{attribute 'linkalways'} 
{attribute 'no_explicit_call' := 'This FB is a CLASS and must be accessed using methods or properties'}
{attribute 'enable_dynamic_creation'}
FUNCTION_BLOCK ABSTRACT NumericDatatypeBase EXTENDS DatatypeBase IMPLEMENTS I_NumericDatatype
VAR
END_VAR

PROPERTY PUBLIC ABSTRACT IsEven : BOOL
GET
END_GET
END_PROPERTY

PROPERTY PUBLIC ABSTRACT IsFloat : BOOL
GET
END_GET
END_PROPERTY

PROPERTY PUBLIC IsOdd : BOOL
GET
IsOdd := not IsEven;
END_GET
END_PROPERTY

PROPERTY PUBLIC ABSTRACT IsSigned : BOOL
GET
END_GET
END_PROPERTY

METHOD PROTECTED OnSerializeTypeWith
VAR_INPUT
	Serializer : I_Serializer;
END_VAR
SUPER^.OnSerializeTypeWith(Serializer);
Serializer.AddKey('minValue');
SerializeMinValue(Serializer);
Serializer.AddKey('maxValue');
SerializeMaxValue(Serializer);
Serializer.AddKeyBool('isSigned', IsSigned);
Serializer.AddKeyBool('isFloat', IsFloat);
END_METHOD

METHOD PROTECTED ABSTRACT SerializeMaxValue
VAR_INPUT
	Serializer : I_Serializer;
END_VAR
END_METHOD

METHOD PROTECTED ABSTRACT SerializeMinValue
VAR_INPUT
	Serializer : I_Serializer;
END_VAR
END_METHOD

END_FUNCTION_BLOCK

(* stored: Version 1.1.0.1, ProductVersion 3.1.4024.13
   POU NumericDatatypeBase: Id {96cfe585-e451-066a-0b8c-26079dae1329}, SpecialFunc None
   Folder Protected: Id {39e73c2d-fc59-01cc-09ba-b5d6d4e55439}
   Property IsEven: Id {f8cc3dde-0e09-0921-2005-35a3a6549198}
   Get Get: Id {ea3f34a8-8bb3-0245-0192-066a15b142d3}
   Property IsFloat: Id {db9b3e2c-dfd9-0457-2028-dc261a7bc18d}
   Get Get: Id {b25b2249-b422-0a33-39c0-da7eeed061cf}
   Property IsOdd: Id {553a9894-a6d5-0755-2f97-e2c62bf116ff}
   Get Get: Id {694de55b-7ecf-07c8-14b2-f6a774a5acba}
   Property IsSigned: Id {c40a7ef2-5152-09e9-260c-22ed7cb9a4b4}
   Get Get: Id {e4a632e5-5d3c-041e-06ba-ac7365bc6ee4}
   Method OnSerializeTypeWith: Id {963c15a2-db3f-0007-3cd1-83c01d967ee1}
   Method SerializeMaxValue: Id {4743dd8e-8f0a-023c-3b23-c1b80869f102}
   Method SerializeMinValue: Id {4191d32a-4a49-06f3-0bae-3e913877ee68} *)
